FUNCTION_BLOCK FB_SaMElementIdle EXTENDS FB_SaMElement
VAR
END_VAR

METHOD FB_init : BOOL
VAR_INPUT
	bInitRetains : BOOL; // if TRUE, the retain variables are initialized (warm start / cold start)
	bInCopyCode : BOOL;  // if TRUE, the instance afterwards gets moved into the copy code (online change)
END_VAR
THIS^.SetText (eLocation := E_BaseLocation.pl, wsDescription := "Bezczynny");
THIS^.SetText (eLocation := E_BaseLocation.en, wsDescription := "Idle");
THIS^.SetText (eLocation := E_BaseLocation.de, wsDescription := "Leerlauf");
THIS^.SetName (stName := THIS^.GetTexts ());
END_METHOD

METHOD PUBLIC InvokeStateForTopElement : BOOL
VAR_INPUT
	itfTopElement		: ITF_BaseSaMStateMethod;
END_VAR
InvokeStateForTopElement	:= itfTopElement.SP_Idle ();
END_METHOD

END_FUNCTION_BLOCK

(* stored: Version 1.1.0.1
   POU FB_SaMElementIdle: Id {8694c703-9934-0e50-2e2e-68f1fa7b47ab}, SpecialFunc None
   Method FB_init: Id {d37b9849-e716-0470-213c-65fb2b59a6b7}
   Method InvokeStateForTopElement: Id {048a8c8a-2009-0cc6-1fe4-6be69c738f1a} *)
